Staubli VAL3: onF6Event.pgx

program onF6Event()
  local num i
  local string l_sItem
begin
  // look if the bButton is enable
  if bButton[5]
    // mark
    // deselect all
    for i=0 to size(sList)-1
      if find(sList[i],"#")!=-1
        sList[i]=right(sList[i],len(sList[i])-1)
      endIf
    endFor
    // select it
    sList[nFrame]="#"+sList[nFrame]
    nFrame=nFrame+1
    use:nView=use:nView+1
  endIf
end
